TYPE ST_IPR_6_1 :
(**************************************************************************************
 * 	Application		:	BoxControl Framework
 *	Revision		:	$Revision: 404529 $
 *	Revision date	:	$Date: 2018-04-23 08:21:38 +0200 (Mo., 23 Apr 2018) $
 *	Last changed by	:	$Author: b7bolm $
 *	URL				:	$URL: http://almscdc.swisslog.com/repo/SWPD/Development/BoxControlFramework/20_Release/trunk/01_Software/BCF/BCF/JumpStart/20_Product/10_App/11_Com/10_Lib/10_Conv/12_MFCS/11_SIS/01_DUTs/11_SIS_6_1/ST_IPR_6_1.TcDUT $
 *
 *	Purpose			:	IPR Structure
 *
 * ------------------------------------------------------------------------------------
 *	Copyright Swisslog [IP AG], Switzerland. All rights reserved.
 * 
 * ------------------------------------------------------------------------------------
 *	
 * 	Revision History: 
 *
 * 	VERSION			DATE			INITIALS			DESCRIPTION
 *	0.1				01.01.2001		swl					Example
 *
 **************************************************************************************)
STRUCT
	Position 			: STRING(SIS_6_1.POSITION_STRINGLENGTH); // 12 Digit SIS Location MM-GGG-EEEE-LLL 
	TU_DataIndex		: STRING(SIS_6_1.TU_DATAINDEX_STRINGLENGTH); // 6 Digit TU-DataIndex 
	MSG_Sequence		: STRING(SIS_6_1.MSG_SEQUENCE_STRINGLENGTH); // 3 Digit Assignment message sequence 
	TU_ID				: STRING(SIS_6_1.TU_ID_STRINGLENGTH); // 18 Digit SSID 
	TU_Type				: STRING(SIS_6_1.TU_TYPE_STRINGLENGTH); // 2 Digit TU-Type 
	AssignmentID		: STRING(SIS_6_1.ASSIGNMENT_ID_STRINGLENGTH); // 8 Digit assignment
	Height				: STRING(SIS_6_1.IPR_HEIGHT_STRINGLENGTH); // 1 Digit Height Result 
	WidthRight			: STRING(SIS_6_1.IPR_WIDTHRIGHT_STRINGLENGTH); // 1 Digit Width Right Result 
	WidthLeft			: STRING(SIS_6_1.IPR_WIDTHLEFT_STRINGLENGTH); // 1 Digit Width Left Result 
	LengthFront			: STRING(SIS_6_1.IPR_LENGTHFRONT_STRINGLENGTH); // 1 Digit Length Front Result 
	LengthRear			: STRING(SIS_6_1.IPR_LENGTHREAR_STRINGLENGTH); // 1 Digit Length Rear Result 
	Weight				: STRING(SIS_6_1.IPR_WEIGHT_STRINGLENGTH); // 7 Digit Weight Value 
	Tunnel				: STRING(SIS_6_1.IPR_TUNNEL_STRINGLENGTH); // 1 Digit Tunnel Result 
	Runner				: STRING(SIS_6_1.IPR_RUNNER_STRINGLENGTH); // 1 Digit Runner Result 
	ErrorCode			: STRING(SIS_6_1.ERRORCODE_STRINGLENGTH); // 4 Digit Scanner Error 
	ValidLabelString	: STRING(SIS_6_1.IPR_VALIDLABELSTRING_STRINGLENGTH); // 3 Digit Valid Label Return Code 
	Label				: STRING(Conveyor.LABEL_LENGTH); // Label Data 
END_STRUCT
END_TYPE

(* stored: Version 1.1.0.1, ProductVersion 3.1.4022.12
   DUT ST_IPR_6_1: Id {a2d71717-b6ae-4d37-b0f7-b6391fb8e790} *)
